Staubli VAL3: RecordJoint.pgx

public program RecordJoint(jointRx& x_j, trsf& x_trTrsf)
  local num l_nNum[2]
begin
  //  $recClean("c")
  //  $recAdd("c","CanIO\Axis8\posCmd_1")
  //  $recAdd("c","CanIO\Axis8\posFbk_1")
  //  $recStart("c",50,250)

  //  $recClean("c")
  //  $recAdd("c","extDrvCmdPos")
  //  $recAdd("c","extDrvCmdVel")
  //  $recAdd("c","extJntCmdPos")
  //  $recAdd("c","extJntCmdVel")
  //  $recAdd("c","extError")
  //  $recAdd("c","extDrvGrpError")
  //  $recStart("c",50,250)

 // x_pPos=$here

 //记录轴的值
  if nAxesSum<1
    popUpMsg("轴个数错误")
    return
  endIf

  resize(nBuffSize,1,nAxesSum)
  x_j=$Xherej(nBuffSize)
  x_trTrsf.x=nBuffSize[0]
  if nAxesSum>1
    x_trTrsf.y=nBuffSize[1]
  endIf

end
